{attribute addProperty BoxType "EL3314-0030-0021"}
{attribute addProperty Id "TC_Inputs_ChannelAT %I*ARRAY[0..3] OF TC_Inputs_Channel_47B3FBFB192240WcStateAT %I*WcState_F855686C1620InfoDataAT %I*InfoData_BC63D37F80100"}
{attribute addProperty CRC "82189946"}
{attribute addProperty SizeInBites "288"}
{attribute addProperty SizeInBytes "36"}
TYPE EL3314_645580BD :
STRUCT
	{attribute addProperty Name "TC_Inputs_Channel"}
	TC_Inputs_Channel : ARRAY[0..3] OF TC_Inputs_Channel_47B3FBFB;
	{attribute addProperty Name "WcState"}
	WcState : WcState_F855686C;
	{attribute addProperty Name "InfoData"}
	InfoData : InfoData_BC63D37F;
END_STRUCT
END_TYPE

(* stored: Version 1.2.0.0, ProductVersion 3.1.4024.9
   DUT EL3314_645580BD: Id {4e2eba48-c689-43aa-9044-234b2a914e46} *)
